Staubli VAL3: initRobotCommandMsg.pgx

program initRobotCommandMsg(RobotCommandMsg& x_msg, bool& x_bError)
begin
  // Copyright 2025 ICUBE Laboratory, University of Strasbourg
  //
  // Licensed under the Apache License, Version 2.0 (the "License");
  // you may not use this file except in compliance with the License.
  // You may obtain a copy of the License at
  //
  //     http://www.apache.org/licenses/LICENSE-2.0
  //
  // Unless required by applicable law or agreed to in writing, software
  // distributed under the License is distributed on an "AS IS" BASIS,
  // WITHOUT WARRANTIES OR CONDITIONS OF ANY KIND, either express or implied.
  // See the License for the specific language governing permissions and
  // limitations under the License.
  x_bError = false

  // Init header fields
  call initHeader(x_msg.header, x_bError)
  if(x_bError == true)
      logMsg("ros2_server::initRobotCommandMsg : Error, failed to init header",2)
      return
  endIf

  // Set message type to RobotCommand (2)
  x_msg.header.nMsgType = 2

  // Total serialized data size = header size + payload size
  x_msg.header.nPayloadSize = 47

  // Resize serialized data buffer
  resize(x_msg.nSerializedData, 1, x_msg.header.nHeaderSize + x_msg.header.nPayloadSize)

  // Resize command data array
  resize(x_msg.robotCommand.nMotionCmdData, 1, 6)

  // Initialize command fields to default values (i.e. STOP command and zeroed data)
  x_msg.robotCommand.nRemoteCtrlPeriod = -1.0
  x_msg.robotCommand.nMotionCmdType = 1
  x_msg.robotCommand.nMotionCmdData[0] = 0.0
  x_msg.robotCommand.nMotionCmdData[1] = 0.0
  x_msg.robotCommand.nMotionCmdData[2] = 0.0
  x_msg.robotCommand.nMotionCmdData[3] = 0.0
  x_msg.robotCommand.nMotionCmdData[4] = 0.0
  x_msg.robotCommand.nMotionCmdData[5] = 0.0

  // Mark message as initialized, but state as not filled
  x_msg.bIsInitialized = true
  x_msg.robotCommand.bIsValid = false

  // OK
  x_bError = false

end
